{attribute 'qualified_only'}
{attribute 'strict'}
TYPE eDCpowerPriority :
(
	auto := 0,
	Inverter := 1,
	DCcoupling	:= 2
);
END_TYPE

(* stored: Version 1.1.0.1, ProductVersion 3.1.4026.18
   DUT eDCpowerPriority: Id {1b854e4d-00df-44d6-ac05-6fb589955ed1} *)
